// Mitsubishi GX Works2 project: 15   PLC: FX3G

// task Task_01 (event TRUE, interval 0, priority 31): POU_01

PROGRAM POU_01
VAR
  wstep : INT;
  wstep2 : INT;
  ton1 : TON;
  wstep3 : INT;
  wstep4 : INT;
  ton2 : TON;
END_VAR
IF M8002 THEN
	wstep := 0;
END_IF;

CASE wstep OF
	0:
		Y0 := FALSE;
		Y1 := FALSE;
		Y2 := FALSE;
		Y3 := FALSE;
		Y4 := FALSE;
		
		IF M10 THEN
			wstep2 := 20;
			wstep3 := 20;
			wstep := 20;
		END_IF;
	
	20:
		Y1 := M8013;
		Y2 := NOT M8013;

		
		IF (wstep2 = 0) AND (wstep3  = 0) THEN
			wstep := 0;
		END_IF;
	
END_CASE;

CASE wstep2 OF
	0:
		Y0 := FALSE;
	
	20:
		Y0 := TRUE;
		ton1(IN := NOT ton1.Q, PT := T#5s);
		IF ton1.Q THEN
			wstep2 := 0;
		END_IF;
END_CASE;

CASE wstep3 OF
	20:
		ton2(IN := NOT ton2.Q, PT := T#2s);
		IF ton2.Q THEN
			wstep3 := 21;
		END_IF;
	
	21:
		Y3 := TRUE;
		ton2(IN := NOT ton2.Q, PT := T#3s);
		IF ton2.Q THEN
			wstep3 := 22;
		END_IF;
		
	22:
		Y3 := FALSE;
		
		Y4 := TRUE;
		ton2(IN := NOT ton2.Q, PT := T#2s);
		IF ton2.Q THEN
			wstep3 := 0;
		END_IF;
END_CASE;
END_PROGRAM
